PROGRAM main_prg
VAR
END_VAR

END_PROGRAM

(* stored: Version 1.1.0.1, ProductVersion 3.1.4024.13
   POU main_prg: Id {051cb0a0-ff0c-4dc6-b4e4-e3d5e458093c}, SpecialFunc None *)
